(* CODESYS project BagAdvanceSequence.xml

Project tree, tasks and I/O mapping:
  function block BagAdvanceSequence [SFC]
*)

// BagAdvanceSequence
FUNCTION_BLOCK BagAdvanceSequence
// This function block is for sequencing the process of advancing
// the next bag forward, allowing the bag time to open with air
// from the blower, and retracting the bag to open with the ice feed shoot.
// If the bag open sensor does not detect that the bag has been 
// opened, the sequence will retry.
// 
// This function does not keep track of the number of attempts, instead
// that count is maintained some level higher than this function. When 
// the bag fails to open, RetryAttempt is pulsed so that the 
// parent function can increment the count.
//
// The higher level function that maintains the failed attempts count
// will pulse the SFCInit input to reset this function back to start.
// The next step then is to seal off the bag and reject it so a new bag
// can be started--that process is managed elsewhere.


VAR_INPUT
	SFCInit: BOOL;
	Trigger: BOOL;
	FirstAdvanceComplete: BOOL;
	FirstRetractComplete: BOOL;
	RetryAdvanceComplete: BOOL;
	RetryRetractComplete: BOOL;
	BagOpen: BOOL;
	ProcessComplete: BOOL;
	CheckOpenDelay: TIME;
	RetryBagOpenDelay: TIME;
END_VAR
VAR_OUTPUT
	FirstAdvance: BOOL;
	FirstRetract: BOOL;
	RetryAttempt: BOOL;
	RetryAdvance: BOOL;
	RetryRetract: BOOL;
	BagReady: BOOL;
END_VAR
VAR
END_VAR

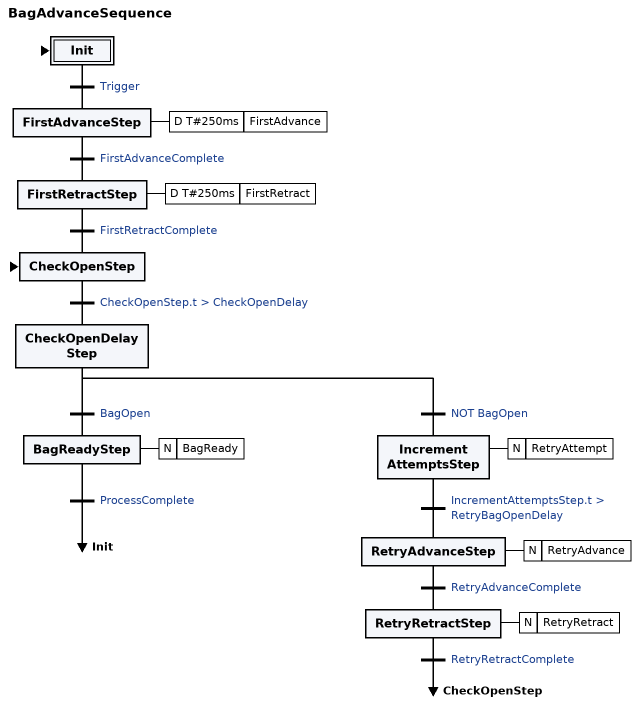
INITIAL_STEP Init:
END_STEP
TRANSITION FROM Init TO FirstAdvanceStep
    := Trigger;
END_TRANSITION
STEP FirstAdvanceStep:
    FirstAdvance(D, T#250ms);
END_STEP
TRANSITION FROM FirstAdvanceStep TO FirstRetractStep
    := FirstAdvanceComplete;
END_TRANSITION
STEP FirstRetractStep:
    FirstRetract(D, T#250ms);
END_STEP
TRANSITION FROM FirstRetractStep TO CheckOpenStep
    := FirstRetractComplete;
END_TRANSITION
STEP CheckOpenStep:
END_STEP
TRANSITION FROM CheckOpenStep TO CheckOpenDelayStep
    := CheckOpenStep.t > CheckOpenDelay;
END_TRANSITION
STEP CheckOpenDelayStep:
END_STEP
TRANSITION FROM CheckOpenDelayStep TO BagReadyStep
    := BagOpen;
END_TRANSITION
TRANSITION FROM CheckOpenDelayStep TO IncrementAttemptsStep
    := NOT BagOpen;
END_TRANSITION
STEP IncrementAttemptsStep:
    RetryAttempt(N);
END_STEP
TRANSITION FROM IncrementAttemptsStep TO RetryAdvanceStep
    := IncrementAttemptsStep.t > RetryBagOpenDelay;
END_TRANSITION
STEP RetryAdvanceStep:
    RetryAdvance(N);
END_STEP
TRANSITION FROM RetryAdvanceStep TO RetryRetractStep
    := RetryAdvanceComplete;
END_TRANSITION
STEP RetryRetractStep:
    RetryRetract(N);
END_STEP
TRANSITION FROM RetryRetractStep TO CheckOpenStep
    := RetryRetractComplete;
END_TRANSITION
STEP BagReadyStep:
    BagReady(N);
END_STEP
TRANSITION FROM BagReadyStep TO Init
    := ProcessComplete;
END_TRANSITION

END_FUNCTION_BLOCK
